{attribute 'linkalways'} 
{attribute 'no_explicit_call' := 'This FB is a CLASS and must be accessed using methods or properties'}
{attribute 'enable_dynamic_creation'}
FUNCTION_BLOCK _ETcVnPixelConnectivity EXTENDS EnumDatatypeBase
VAR
	localData : ETcVnPixelConnectivity;
	activeData : REFERENCE TO ETcVnPixelConnectivity;
	enumBaseDatatype : _DINT(localData);
END_VAR

METHOD PRIVATE AddLocalEnumeration
VAR_INPUT
	Enumeration : T_MAXSTRING;
	Value : ETcVnPixelConnectivity;
END_VAR
AddEnumeration(Enumeration, Value);
END_METHOD

PROPERTY PUBLIC Address : PVOID
GET
Address := ADR(activeData);
END_GET
END_PROPERTY

METHOD PUBLIC ClearReference
VAR_INPUT
END_VAR
activeData REF= localData;
SetBaseDatatypeReference();
END_METHOD

METHOD PUBLIC Clone : I_Datatype
VAR
    pClone : POINTER TO _ETcVnPixelConnectivity;
END_VAR
pClone := __NEW(_ETcVnPixelConnectivity(InitialValue := Value));
Clone := pClone^;
END_METHOD

METHOD FB_init : BOOL
VAR_INPUT
	bInitRetains : BOOL; // if TRUE, the retain variables are initialized (warm start / cold start)
	bInCopyCode : BOOL;  // if TRUE, the instance afterwards gets moved into the copy code (online change)
	InitialValue : ETcVnPixelConnectivity;
END_VAR
localData := InitialValue;
AddBaseDatatype(enumBaseDatatype);
ClearReference();

AddLocalEnumeration('TCVN_PC_4', ETcVnPixelConnectivity.TCVN_PC_4);
AddLocalEnumeration('TCVN_PC_8', ETcVnPixelConnectivity.TCVN_PC_8);
END_METHOD

PROPERTY PUBLIC Identifier : T_MAXSTRING
GET
Identifier := 'ETcVnPixelConnectivity';
END_GET
END_PROPERTY

METHOD IsEnumeratorValueEqual : BOOL
VAR_INPUT
	Enumerator : I_KeyValueForwardEnumerator;
END_VAR
VAR
	storedValue : ETcVnPixelConnectivity;
END_VAR
IF NOT Enumerator.TryGet(storedValue) THEN
	RETURN;
END_IF

IsEnumeratorValueEqual := storedValue = activeData;
END_METHOD

METHOD PUBLIC MakeReferenceTo
VAR_INPUT
	ReferenceTarget : REFERENCE TO ETcVnPixelConnectivity;
END_VAR
activeData REF= ReferenceTarget;
SetBaseDatatypeReference();
END_METHOD

METHOD PROTECTED SetBaseDatatypeReference
VAR_INPUT
END_VAR
enumBaseDatatype.MakeReferenceTo(activeData);
END_METHOD

PROPERTY PUBLIC Size : UDINT
GET
Size := SIZEOF(activeData);
END_GET
END_PROPERTY

METHOD TryMakeReferenceTo : BOOL
VAR_INPUT
	Target : I_Datatype;
END_VAR
VAR
	targetAsEnum : I_EnumDatatype;
	pTargetData : POINTER TO ETcVnPixelConnectivity;
END_VAR
IF NOT Target.TryResolveAsEnumDatatype(targetAsEnum) THEN
	RETURN;
END_IF

IF targetAsEnum.Identifier <> Identifier THEN
	RETURN;
END_IF

pTargetData := Target.Address;
activeData REF= pTargetData^;
SetBaseDatatypeReference();
TryMakeReferenceTo := TRUE;
END_METHOD

PROPERTY PUBLIC Value : ETcVnPixelConnectivity
GET
Value := activeData;
END_GET
SET
activeData := Value;
END_SET
END_PROPERTY

END_FUNCTION_BLOCK

(* stored: Version 1.1.0.1, ProductVersion 3.1.4024.12
   POU _ETcVnPixelConnectivity: Id {00d7e4fe-0919-0d89-1765-aec693ce9d92}, SpecialFunc None
   Folder Constructor: Id {208f36ac-7f83-027b-13cf-fddb87a340f2}
   Folder Private: Id {7478ad53-ff7d-015a-1ce5-03f65c107ed9}
   Folder Protected: Id {8eee0925-cc27-0b3c-234c-7a2344437599}
   Method AddLocalEnumeration: Id {611aed11-379c-02da-3c15-21d9f424bae9}
   Property Address: Id {945c44a8-5f59-0549-3fe6-a06fdd15b979}
   Get Get: Id {efd156d0-7560-04dc-2ba3-08a834871d1e}
   Method ClearReference: Id {acf8e8ab-76b8-0b3b-3748-a32e8f367da7}
   Method Clone: Id {2cd5d6a7-9217-05df-00c8-7273226e0161}
   Method FB_init: Id {718405cb-445a-0e58-2a6e-4f98b4dfa2a7}
   Property Identifier: Id {347a1130-88a6-057f-1979-4f27431e1aa0}
   Get Get: Id {91426f67-ca7a-0e58-3686-aa2f7b19d417}
   Method IsEnumeratorValueEqual: Id {87ca2e3a-62af-01fe-0e2b-e7914c6e85d7}
   Method MakeReferenceTo: Id {24625d42-60b3-0202-3ff9-9b20aa2d7c8b}
   Method SetBaseDatatypeReference: Id {c8524817-847b-0379-2179-7168f67b0730}
   Property Size: Id {f099b73d-d78c-00c0-3f57-3f3626d7d966}
   Get Get: Id {b8e5a7be-7778-0e17-3eb9-b3de12ae4807}
   Method TryMakeReferenceTo: Id {6906f907-d4b7-03bf-08fb-b89b17d834d7}
   Property Value: Id {71f06e9d-9e8d-0c0a-3369-6878f6f03e1f}
   Get Get: Id {d56f4e0b-7a24-0ae8-3e9e-6e0e38518a1b}
   Set Set: Id {08e1d0c1-92ed-0a9a-2d3f-415274f016ab} *)
